(*
Nazwa:			FB_EntranceGatesFesto
Opis:			Stacja szlabanów do przesuwania formatek	
Wersja:			v1.1
Data:			2020-09-30
Autor:			DP
Urzadzenia:		do 1 szlabanu na siłowniku beckhoff i 1 szlabanu zatrzymującego na końcu
Konfiguracja:	
Info: 
*)
FUNCTION_BLOCK FB_EntranceGatesServo
VAR_INPUT
	bEnable						:BOOL;			//Zezwolenie na pracę
	bEStop						:BOOL;			//Stop Awaryjny włączony
	bRunPrepare					:BOOL;			//Rozkaz przesuwania formatek do środka 
	bRun						:BOOL;			//Rozkaz wpuszczenia dwóch formatek 
	bHoming						:BOOL;			//Zezwolenie na wykonanie bazowania i pozycjonowania podajnika
	bHeightSet					:BOOL;			//Ustaw wysokość
	bIgnoreError				:BOOL;			//Ignorowania błędów cyklu pracy
	bReset						:BOOL;			//Reset błędu, jeśli w stanie "eError"
	bBlocking					:BOOL;			//Blokowanie pierwszego szlabanu

	bOpenedGate1ActuatorSensor	:BOOL;			//Czujnik otwarcia siłownika szlabanu 1
	bOpenedGate2ActuatorSensor	:BOOL;			//Czujnik otwarcia siłownika szlabanu 2
	bClosedGate1ActuatorSensor	:BOOL;			//Czujnik zamknięcia siłownika szlabanu 1
	bClosedGate2ActuatorSensor	:BOOL;			//Czujnik zamknięcia siłownika szlabanu 2
	bMovingTwoForms				:BOOL;			//Przesuwanie o dwie formatki
	bMovingThreeForms			:BOOL;			//Przesuwanie o trzy formatki
	bManualMovement				:BOOL;			//Zezwolenie na ruchy ręcznę
	bHomingStateGate1			:BOOL;			//Stan bazowania szlabanów nr 1
	bHomingStateGate2			:BOOL;			//Stan bazowania szlabanów nr 2
	bResetState					:BOOL;			//Resetowanie stanu stacji

	//Parametry przeciągania formatek

	lrPullReadyPosition			:LREAL;			//Pozycja przeciągania przy starcie dozowania
	lrPullStopOnePhasePosition	:LREAL;			//Pozycja stopu przeciągania przy dozowaniu jednofazowym
	lrPullStopTwoPhasePosition	:LREAL;			//Pozycja stopu przeciągania przy dozowaniu dwufazowym
	lrPullVelocity				:LREAL;			//Prędkość przeciągania 
	lrPullAcceleration			:LREAL;			//Przyśpieszenie przeciągania
	lrPullDeceleration			:LREAL;			//Zwalnianie przeciągania
	
	_ALARMINFO_					:BOOL;
	iStationIndex				:UDINT;			//Numer stacji 
	sStationName				:STRING;		//Nazwa stacji

END_VAR
VAR_OUTPUT
	
	eState						:E_Station;				//Stan ogólny bloku
	eRunningState				:E_EntranceGatesState;	//Stan szlabanów
	bError						:BOOL;					//Błąd stacji	
	nErrorNr					:UDINT;					//Nr błędu podajnika platynek
	sErrorDescription			:STRING(200);			//Opis błędu
	sErrorDescription2			:STRING(200);			//Opis błędu
	sErrorStationName			:STRING;				//Nazwa stacji
	bGate1Actuator				:BOOL;					//Sterownie siłownika szlabanu 1
	bGate2Actuator				:BOOL;					//Sterownie siłownika szlabanu 2
	tCycleTime					:TIME;
	bHomingDone					:BOOL;					//Wymagane ponowne bazowanie (blad podczas bazowania lub stop awaryjny)
	bCyclePrepareDone			:BOOL;
	bCycleDone					:BOOL;
	bCycleNotDone				:BOOL;
	//WEJSCIA WYJSCIA SPRZETOWE
	nPullServoErrorNr			:UDINT;
	lrPullActualPosition		:LREAL;

END_VAR

VAR

	(**********BECKHOFF PRZECIAGANIE******************)
	mcPullMoveAbsolute			:MC_MoveAbsolute; 	// Blok nr 1 ruchu absolutnego tłoka dozownika
	mcPullManualMove			:MC_JOG;			// Blok ruchu manualnego tłokiem dozownika
	mcPullStop					:MC_Stop;			// Blok zatrzymania tłoka dozownika, jeśli to konieczne
	mcPullSoftReset				:MC_Reset;			// Blok łagodnego resetu serwa tloka dozownika
	mcPullPower					:Mc_Power;			// Blok zasilania serwa dozownika
	bPullServoPower				:BOOL; 				// Zalaczenie zasilania serwa
	// Blok resetowania twardego błędu
	fbPullHardReset				:FB_SoEReset;
	bStopped					:BOOL;
		
	// Timer blokady otwierania chwytaka
	tonOpeningGate1Blocked		:TON;
	tonOpeningGate2Blocked		:TON;
	tonClosingGate1Blocked		:TON;
	tonClosingGate2Blocked		:TON;
	tonCycleTimer				:TON;
	rtrigCycleTimerRead			:R_TRIG;	
	bLastStateGate1Actuator		:BOOL;
	bLastStateGate2Actuator		:BOOL;	
	eLastState					:E_Station;				//Stan ogólny bloku
	eLastRunningState			:E_EntranceGatesState;	//Stan podbloku
	eLastStateTemp				:E_Station;				//Stan ogólny bloku
	eLastRunningStateTemp		:E_EntranceGatesState;	//Stan podbloku

	bStateError: BOOL;
		rtPulling: R_TRIG;
	rtPreparingToReady: R_TRIG;
	rtPullingToMiddle: R_TRIG;
	tonDelayServoOn			: TON;

	bNotPreapreToReadyAfterEstop: BOOL;
	lrtest: LREAL;
	tonGate1Actuator: TON;
END_VAR

VAR_IN_OUT
	bManualGate1Actuator	:BOOL;			//Ruch ręczny siłownikiem szlabanu 1
	bManualGate2Actuator	:BOOL;			//Ruch ręczny siłownikiem szlabanu 2
	bManualPullLeft			:BOOL;			//Ruch ręczny przeciąganiem w lewo
	bManualPullRight		:BOOL;			//Ruch ręczny przeciąganiem w prawo
	PullAxisRef				:AXIS_REF;		//Struktura sterowania NC dla serwa zakręcania
END_VAR

(*Przepisywanie Homingu , rozdzielenie wyjść*)

ErrorHandling();
Control();
GatesControlBlocks();
Statistics();


(*wypracowanie sygnałów wyjściowych z bloku*)
lrPullActualPosition:=PullAxisRef.NcToPlc.ActPos;	//Pozycja 


(*Zapisywanie ostatniego stanu*)
IF eLastStateTemp<>eState THEN
	eLastState := eLastStateTemp;
END_IF
eLastStateTemp := eState;
IF eLastRunningStateTemp<>eRunningState THEN
	eLastRunningState := eLastRunningStateTemp;
END_IF
eLastRunningStateTemp := eRunningState;

(*Koniec Zapisywanie ostatniego stanu*)



IF bResetState AND NOT bBlocking THEN
	eState:=E_Station.eReady;
	eRunningState:=eLastRunningState:=E_EntranceGatesState.eReady;
	bGate1Actuator:=bHomingStateGate1;
	bGate2Actuator:=bHomingStateGate2;
END_IF

ACTION Control:

	(** TIMERY**)
	rtPulling(CLK:=eRunningState=E_EntranceGatesState.ePulling AND bOpenedGate1ActuatorSensor AND bClosedGate2ActuatorSensor, Q=>);
	rtPullingToMiddle(CLK:=eRunningState=E_EntranceGatesState.ePullingToMiddle AND bOpenedGate1ActuatorSensor AND bClosedGate2ActuatorSensor, Q=>);
	rtPreparingToReady(CLK:=eRunningState=E_EntranceGatesState.ePreparingToReady AND bClosedGate1ActuatorSensor, Q=>);
	
	tonDelayServoOn(IN:=(eState = E_Station.ePreparingToReady), PT:=T#1200MS);
	tonGate1Actuator(IN:=bGate1Actuator, PT:=T#100MS); // Opóżnienie sygnału wyjścia pierwszego szlabany, uzyte do opoznienia wylaczania drugiego
	(*****Wyłączenie enable*****)
	IF NOT bEnable THEN
		IF eState <> E_Station.eDisabled AND eState <> E_Station.ePreparingToDisable THEN
				eState 				:= E_Station.ePreparingToDisable; 
		END_IF	
	END_IF

	(*****Estop*****)
	IF NOT bEstop  THEN	
		IF eState <> E_Station.eAborted AND eState <> E_Station.eAborting AND eState <> E_Station.eDisabled THEN
				eState 				:= E_Station.eAborting; 
		END_IF
	END_IF

	
	CASE eState OF
	/////////////////////////////	
		E_Station.eDisabled: 					// Stan nieaktywnosci (Stacja wyłączona) 
		
			IF bEnable THEN
				eState 				:= E_Station.ePreparingToReady; 
			END_IF 
			
    /////////////////////////////	    
		E_Station.eAborted: 					// Stan bezpiecznego zatrzymania (po Abortingu) 

			IF bEStop THEN
				eState 				:= E_Station.ePreparingToReady;
			END_IF
			
	/////////////////////////////	
		E_Station.eAborting:                 	// Stan bezpiecznego zatrzymywania (po EStopie)

		mcPullManualMove.JogBackwards		:=	FALSE;
		mcPullManualMove.JogForward			:=	FALSE;
		mcPullMoveAbsolute.Execute 			:=	FALSE;
		
		//bPullServoPower						:=	TRUE;
		mcPullPower.Override				:=	100;		
		mcPullStop.Execute					:=	NOT bStopped;
		bNotPreapreToReadyAfterEstop		:= TRUE;
		IF (mcPullStop.Done OR mcPullStop.Error OR bStopped) THEN
			bStopped						:=	FALSE;
			bPullServoPower					:=	FALSE;
			mcPullStop.Execute				:=	FALSE;
			eLastRunningState				:=	eRunningState;
			eRunningState					:= E_EntranceGatesState.eReady;
			eState 							:=	E_Station.eAborted; 
		END_IF
			
	/////////////////////////////			
		E_Station.eError:                 	 	// Stan błędu 	
	
			mcPullMoveAbsolute.Execute 			:=	FALSE;
			mcPullStop.Execute					:= FALSE;
			IF bReset THEN
				eState 							:=	E_Station.eResetting;
			ELSE
				mcPullSoftReset	(Execute:=FALSE,Axis:=PullAxisRef);		
			END_IF
			
	/////////////////////////////
		E_Station.eResetting:					// Stan resetowania bledu (po Errorze)
			
			//Procedura obsługi resetu w zależności od błędu
			CASE nErrorNr-iStationIndex OF
		
				//Error 1 - ZACIETY SZLABAN
				1:
					bGate1Actuator								:=	FALSE;		
					nErrorNr									:=	0;
					bError										:=	FALSE;
					sErrorDescription							:=	'';		
					
				//Error 8 - SZLABANYW ZŁEJ POZYCJI			
				8: 
					bGate1Actuator								:=	FALSE;		
					bGate2Actuator								:=	TRUE;		// z 17.11.2020
				//IF tonDelayServoOn.Q THEN
					bPullServoPower								:=	TRUE;
				//END_IF
					IF bClosedGate1ActuatorSensor AND mcPullPower.Status THEN	
						mcPullMoveAbsolute.Velocity			:= lrPullVelocity;
						mcPullMoveAbsolute.Position			:= lrPullReadyPosition;
						mcPullMoveAbsolute.Acceleration		:= 15000;
						mcPullMoveAbsolute.Deceleration		:= 15000;
						mcPullMoveAbsolute.Execute			:= TRUE;
					
						//Wykonano ruch
						IF mcPullMoveAbsolute.Done THEN
							mcPullMoveAbsolute.Execute 		:=	FALSE;
							bError := FALSE;
						END_IF		
					END_IF
				//Error 9, Error 10 - BŁĄD SERWA PRZECIAGANIA
				9,10:	
					fbPullHardReset(Execute:=NOT mcPullMoveAbsolute.Execute,Axis:=PullAxisRef);
					mcPullSoftReset(Execute:=TRUE,Axis:=PullAxisRef);																		
					(*IF NOT fbPullHardReset.Busy AND NOT mcPullSoftReset.Busy AND mcPullPower.Status AND NOT PullAxisRef.Status.Error THEN
						fbPullHardReset(Execute:=FALSE,Axis:=PullAxisRef);
						mcPullSoftReset(Execute:=FALSE,Axis:=PullAxisRef);
						mcPullMoveAbsolute.Execute:=TRUE;
						mcPullMoveAbsolute.Position:=lrPullReadyPosition; 
						IF mcPullMoveAbsolute.Done=TRUE THEN
							mcPullMoveAbsolute.Execute:=FALSE;
							nErrorNr:=0;
							nPullServoErrorNr:=0;
							mcPullPower.Override:=100;
							bError := FALSE;
							sErrorDescription:='';	
						END_IF*)
					IF NOT fbPullHardReset.Busy AND NOT mcPullSoftReset.Busy (*AND NOT mcPullPower.Status*) AND NOT PullAxisRef.Status.Error  THEN
						fbPullHardReset(Execute:=FALSE,Axis:=PullAxisRef);
						mcPullSoftReset(Execute:=FALSE,Axis:=PullAxisRef);
						nPullServoErrorNr:=0;
						nErrorNr:=0;
						mcPullPower.Override:=100;
						bError := FALSE;
						sErrorDescription:='';			  	
					END_IF
					
				ELSE
					bError := FALSE;	
	
				END_CASE	
			
			IF NOT bError THEN
				nErrorNr 			:=	0;
   				sErrorDescription 	:=	'';
   				sErrorDescription2 	:=	'';	
				eState 				:=	E_Station.ePreparingToReady;
			ELSE
				eState 				:=	E_Station.eError;
			END_IF
        
	/////////////////////////////
		E_Station.eManualMovement:     			// Stan ruchów manualnych  
       
			ManualMovements();
			//Wyjście z trybu serwisowego
			IF NOT bManualMovement THEN
				
				bGate1Actuator:=bLastStateGate1Actuator;
				bGate2Actuator:=bLastStateGate2Actuator;
	
				//Ruch 
				mcPullPower.Override				:= 100;
				mcPullMoveAbsolute.Velocity			:= lrPullVelocity;
				mcPullMoveAbsolute.Position			:= lrPullReadyPosition;
				mcPullMoveAbsolute.Acceleration		:= 1000;
				mcPullMoveAbsolute.Deceleration		:= 1000;
				mcPullMoveAbsolute.Execute			:= TRUE;
			
				//Wykonano ruch
				IF mcPullMoveAbsolute.Done THEN
					mcPullMoveAbsolute.Execute 		:=	FALSE;
					eState							:=	E_Station.eReady;
					eRunningState					:=	E_EntranceGatesState.eReady;
				END_IF
				
			END_IF

	/////////////////////////////
		E_Station.eHoming:						// Stan bazowania 

			Homing();
			IF NOT bHoming AND NOT bHeightSet THEN
			   eState							:=	E_Station.ePreparingToReady;
			   mcPullManualMove.JogForward		:=	FALSE;
			   mcPullManualMove.JogBackwards	:=	FALSE;
			END_IF		
			
	/////////////////////////////
		E_Station.eHomingDone:                  // Stan wykonania bazowania 
		
			mcPullManualMove.JogForward			:=	FALSE;
			mcPullManualMove.JogBackwards		:=	FALSE;
			bHomingDone							:=	TRUE;
			IF NOT bHoming AND NOT bHeightSet THEN
			   eState:=E_Station.eReady;
			END_IF
			
	/////////////////////////////
		E_Station.ePreparingToReady:            // Stan przygotowywania do gotowosci (zawsze przed Ready)  
		
		eRunningState						:=	E_EntranceGatesState.eReady;
		IF NOT bNotPreapreToReadyAfterEstop THEN //LastRunningState przypisuje w abborting
			bGate1Actuator								:=	FALSE;		
			bGate2Actuator								:=	TRUE;		// z 17.11.2020
			IF tonDelayServoOn.Q THEN
				bPullServoPower								:=	TRUE;
			END_IF
			IF bClosedGate1ActuatorSensor AND mcPullPower.Status THEN
				IF bHomingDone THEN		
					mcPullMoveAbsolute.Velocity			:= lrPullVelocity;
					mcPullMoveAbsolute.Position			:= lrPullReadyPosition;
					mcPullMoveAbsolute.Acceleration		:= 15000;
					mcPullMoveAbsolute.Deceleration		:= 15000;
					mcPullMoveAbsolute.Execute			:= TRUE;
				
					//Wykonano ruch
					IF mcPullMoveAbsolute.Done THEN
						mcPullMoveAbsolute.Execute 		:=	FALSE;
						eRunningState					:=	E_EntranceGatesState.eReady;
						eState							:=	E_Station.eReady;	
					END_IF
								
				ELSIF NOT bHomingDone THEN
					eRunningState						:=	E_EntranceGatesState.eReady;
					eState								:=	E_Station.eReady;	
				END_IF
			END_IF
		ELSE //estop byl trakcie
			IF tonDelayServoOn.Q THEN
				bPullServoPower								:=	TRUE;
			END_IF
			IF  mcPullPower.Status THEN
				//bNotPreapreToReadyAfterEstop				:= FALSE;
				eState										:=	E_Station.eReady;	
				//eRunningState								:=	eLastRunningState; //Wpisze ostatni stan
			END_IF
		END_IF
			
	/////////////////////////////
		E_Station.ePreparingToDisable:          // Stan przygotowywania do nieaktywnosci (po wyłączeniu Enable) 
  
			bGate1Actuator							:=	FALSE;		
			bGate2Actuator							:=	FALSE;		
			bPullServoPower							:=	TRUE;
			
			IF mcPullPower.Status THEN
				mcPullPower.Override				:=	10;
				mcPullMoveAbsolute.Velocity			:=	100;
				mcPullMoveAbsolute.Execute			:=	TRUE;
				mcPullMoveAbsolute.Position			:=	lrPullReadyPosition;
				IF mcPullMoveAbsolute.Done THEN
					mcPullMoveAbsolute.Execute 		:=	FALSE;
					eState							:=	E_Station.eDisabled;
					eRunningState					:=	E_EntranceGatesState.eReady;
				END_IF	
			END_IF
			
			IF bIgnoreError THEN
				eState								:=	E_Station.eDisabled;
				eRunningState						:=	E_EntranceGatesState.eDisabled;
			END_IF
			
	/////////////////////////////
		E_Station.eReady:						// Stan gotowosci 
		
			IF (bRunPrepare OR bRun) AND NOT bCycleDone AND NOT bCycleNotDone THEN
				eState 				:= E_Station.eStarting; 
			END_IF
			IF bHoming OR bHeightSet THEN
				eState 				:= E_Station.eHoming; 
			END_IF
			IF bManualMovement THEN
				//Jeśli przejście w tryb ruchów manualnych przepisz wszystkie stany siłowników sterowanych przez moduł
				//aby zapobiec ewentualnym kolizjom po wejściu w tryb serwisowy
				bLastStateGate1Actuator		:=	bGate1Actuator;
				bLastStateGate2Actuator		:=	bGate2Actuator;
				bManualGate1Actuator		:=	bGate1Actuator;
				bManualGate2Actuator		:=	bGate2Actuator;				
				eState 						:=	E_Station.eManualMovement; 
			END_IF
			IF NOT bRun THEN
				bCycleDone 					:= FALSE;
				bCycleNotDone 				:= FALSE;	
				bCyclePrepareDone			:= FALSE;		
			END_IF
			
			bStopped						:= FALSE;
			mcPullStop.Execute				:= FALSE;
			
	/////////////////////////////
		E_Station.eStopping:					// Stan zatrzymywania 


			Running();		
			
			mcPullStop.Execute				:=	NOT bStopped;

			IF (mcPullStop.Done OR mcPullStop.CommandAborted) THEN
				 bStopped					:=	TRUE;
			END_IF
			
			IF bStopped AND NOT mcPullStop.Execute THEN
				eState 						:=	E_Station.eReady;	
			END_IF
			

	/////////////////////////////
		E_Station.eStarting:                  	// Stan uruchamiania (po Ready)
		
			eState					 := E_Station.eRunning; 
			
	/////////////////////////////
		E_Station.eRunning:               		// Stan wykonywania cyklu (po Startingu), w tym stanie osobny
 
			IF 	bNotPreapreToReadyAfterEstop THEN //Zmiana 17112020
				bNotPreapreToReadyAfterEstop := FALSE;
				eRunningState								:=	eLastRunningState; //Wpisze ostatni stan
			END_IF
		
			Running();
			IF NOT bRun AND NOT bRunPrepare THEN					(*Przerywanie cyklu*)
				eState 				 := E_Station.eStopping;	
			END_IF
			IF bCycleDone OR bCycleNotDone THEN (*Cykl zakończony*)
				//eState 				 := E_Station.eReady;//Zmiana
				eState 				 := E_Station.ePreparingToReady;
			END_IF	
			
	/////////////////////////////		
	END_CASE
END_ACTION

ACTION ErrorHandling:
//OBSŁUGA BŁĘDÓW PODAJNIKA PLATYNEK

//************LISTA BŁĘDÓW***************
bStateError:= (eState=E_Station.eError) OR (eState=E_Station.eResetting);

IF bEnable THEN

	//Error 1 - Blokada otwarcia szlabanu wejściowego nr 1
	tonOpeningGate1Blocked(IN:= bGate1Actuator AND NOT bOpenedGate1ActuatorSensor, PT:=T#2S);
	IF tonOpeningGate1Blocked.Q AND NOT bStateError THEN
		sErrorDescription:='Blokada otwarcia szlabanu wjazdowego nr 1 - sprawdź czujnik lub odblokuj mechanicznie';
		bError := TRUE;
		nErrorNr:=1;	
		nErrorNr:=nErrorNr+iStationIndex;
	END_IF
	
	//Error 2 - Blokada otwarcia szlabanu wejściowego nr 2
	tonOpeningGate2Blocked(IN:= bGate2Actuator AND NOT bOpenedGate2ActuatorSensor, PT:=T#2S);
	IF tonOpeningGate2Blocked.Q AND NOT bStateError THEN
		sErrorDescription:='Blokada otwarcia szlabanu wjazdowego nr 2 - sprawdź czujnik lub odblokuj mechanicznie';
		bError := TRUE;
		nErrorNr:=2;	
		nErrorNr:=nErrorNr+iStationIndex;
	END_IF
				
	//Error 4 - Blokada zamknięcia szlabanu wejściowego nr 1
	tonClosingGate1Blocked(IN:= NOT bGate1Actuator AND NOT bClosedGate1ActuatorSensor, PT:=T#2S);
	IF tonClosingGate1Blocked.Q AND NOT bStateError THEN
		sErrorDescription:='Blokada zamknięcia szlabanu wjazdowego nr 1 - sprawdź czujnik lub odblokuj mechanicznie';
		bError := TRUE;
		nErrorNr:=2;	
		nErrorNr:=nErrorNr+iStationIndex;
	END_IF

	//Error 5 - Blokada zamknięcia szlabanu wejściowego nr 2
	tonClosingGate2Blocked(IN:= NOT bGate2Actuator AND NOT bClosedGate2ActuatorSensor, PT:=T#2S);
	IF tonClosingGate2Blocked.Q AND NOT bStateError THEN
		sErrorDescription:='Blokada zamknięcia szlabanu wjazdowego nr 2 - sprawdź czujnik lub odblokuj mechanicznie';
		bError := TRUE;
		nErrorNr:=2;	
		nErrorNr:=nErrorNr+iStationIndex;
	END_IF	
		
(*	//Error 8 - SZLABANY W ZŁEJ POZYCJI
	IF (ABS(PullAxisRef.NcToPlc.ActPos) - lrPullReadyPosition) > 5 AND bHomingDone AND eState = E_Station.eReady AND NOT bResetState AND NOT bStateError THEN
		bError := TRUE;
		nErrorNr:=8;
		nErrorNr:=nErrorNr+iStationIndex;
		nPullServoErrorNr:=PullAxisRef.Status.ErrorID;
		sErrorDescription:='Szlabany w złej pozycji, zresetuj';
		sErrorDescription2:=INT_TO_STRING(LREAL_TO_INT(PullAxisRef.NcToPlc.ActPos));
	END_IF;	*)
	
	//Error 9 - BŁĄD SERWA PODNOSZENIA ZAKRĘCARKI
	IF (PullAxisRef.Status.Error OR mcPullPower.Error) AND NOT bStateError THEN
		bError := TRUE;
		nErrorNr:=9;
		nErrorNr:=nErrorNr+iStationIndex;
		nPullServoErrorNr:=PullAxisRef.Status.ErrorID;
		sErrorDescription:='Błąd napędu przeciągania Błąd NC:';
		sErrorDescription2:=F_AxErrMsg(nPullServoErrorNr);
	END_IF;	
	
	//Error 10 - BŁĄD INNY SERWA PODNOSZENIA ZAKRĘCARKI
	IF  mcPullMoveAbsolute.Error AND NOT bStateError THEN
		bError := TRUE;
		nErrorNr:=10;
		nErrorNr:=nErrorNr+iStationIndex;
		nPullServoErrorNr:=mcPullMoveAbsolute.ErrorID;
		sErrorDescription:='Błąd napędu przeciągania Błąd NC:';
		sErrorDescription2:=F_AxErrMsg(nPullServoErrorNr);
	END_IF;
	
	
	
ELSE
	bError := FALSE;
END_IF
	
//*******KONIEC LISTA BŁĘDÓW***************	

	

//******************PRZEJŚCIE DO eERROR*****************************

IF bError AND NOT bStateError THEN
	IF eLastState = eRunning THEN
		bCycleNotDone := TRUE;
	END_IF
	eState := E_Station.eError;
END_IF

//****************WYŚWIETLANIE STATUSU BLEDU***********************


(*Wyświetlanie błedu na wyjściu*)
bError;

(*Przepisywanie nazwy stacji*)
sErrorStationName:=sStationName;
END_ACTION

ACTION GatesControlBlocks:
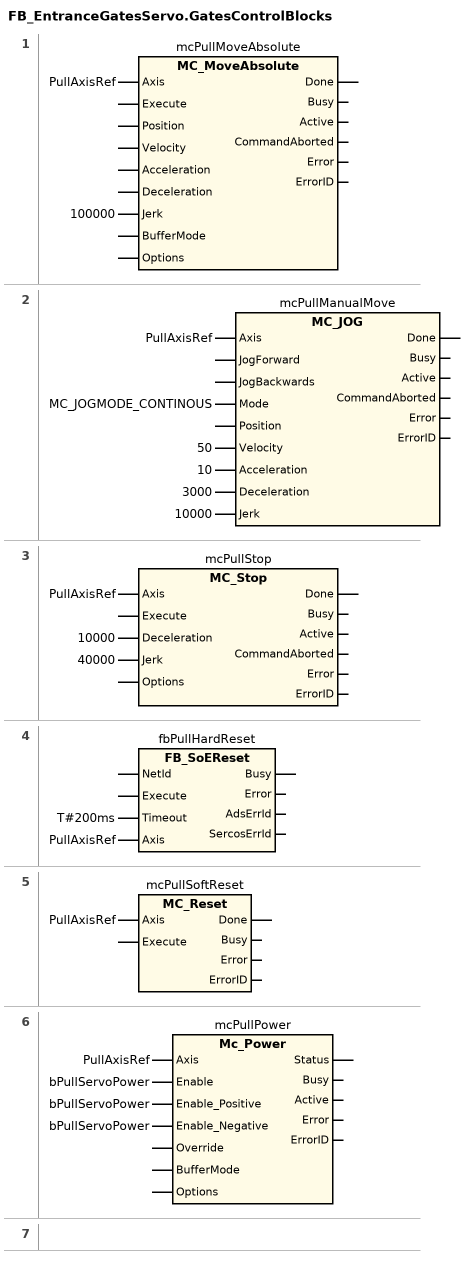
// NETWORK 1
mcPullMoveAbsolute(Axis := PullAxisRef, Jerk := 100000); // MC_MoveAbsolute

// NETWORK 2
mcPullManualMove(
    Axis := PullAxisRef,
    Mode := MC_JOGMODE_CONTINOUS,
    Velocity := 50,
    Acceleration := 10,
    Deceleration := 3000,
    Jerk := 10000); // MC_JOG

// NETWORK 3
mcPullStop(Axis := PullAxisRef, Deceleration := 10000, Jerk := 40000); // MC_Stop

// NETWORK 4
fbPullHardReset(Timeout := T#200ms, Axis := PullAxisRef); // FB_SoEReset

// NETWORK 5
mcPullSoftReset(Axis := PullAxisRef); // MC_Reset

// NETWORK 6
mcPullPower(
    Axis := PullAxisRef,
    Enable := bPullServoPower,
    Enable_Positive := bPullServoPower,
    Enable_Negative := bPullServoPower); // Mc_Power

// NETWORK 7
END_ACTION

ACTION Homing:
//Ustawienia początkowe
bGate1Actuator						:=	FALSE;
bGate2Actuator						:=	TRUE;

//Włączanie zasilania
mcPullPower.Override				:=	100;
mcPullManualMove.JogBackwards		:=	FALSE;
mcPullManualMove.JogForward			:=	FALSE;
bPullServoPower						:=	TRUE;

//Serwo włączone
IF mcPullPower.Status THEN
	
	//Ruch 
	mcPullMoveAbsolute.Velocity			:= lrPullVelocity;
	mcPullMoveAbsolute.Position			:= lrPullReadyPosition;
	mcPullMoveAbsolute.Acceleration		:= 1000;
	mcPullMoveAbsolute.Deceleration		:= 1000;
	mcPullMoveAbsolute.Execute			:= TRUE;

	//Wykonano ruch
	IF mcPullMoveAbsolute.Done THEN
		mcPullMoveAbsolute.Execute 		:=	FALSE;
		eState							:=	E_Station.eHomingDone;
	END_IF
END_IF
END_ACTION

ACTION ManualMovements:

//W trybie ruchów manualnych wykonuj ruchy za pomocą rozkazów manualnych
IF NOT bRun AND NOT bRunPrepare THEN
	bGate1Actuator					:=	bManualGate1Actuator;
	bGate2Actuator					:=	bManualGate2Actuator;	
	mcPullPower.Override			:=	100;
	mcPullManualMove.JogForward		:=	bManualPullRight;
	mcPullManualMove.JogBackwards	:=	bManualPullLeft;
ELSE	
	;
END_IF


IF bHoming OR bHeightSet THEN
	eState:=E_Station.eHoming;
END_IF
	

Running();


IF NOT bRun AND NOT bRunPrepare THEN
	bCycleDone 					:= FALSE;
	bCycleNotDone 				:= FALSE;			
	bCyclePrepareDone			:= FALSE;
END_IF
END_ACTION

ACTION Running:


CASE eRunningState OF
	
	//NIEGOTOWY
	E_EntranceGatesState.eDisabled:
			eRunningState:=E_EntranceGatesState.eReady;
		
	//ZGRZEWANIE GOTOWY DO PRACY
	E_EntranceGatesState.eReady:
		
		//Jeśli komenda podania platynki przejdź do stanu zasysania platynki
		IF NOT bCycleDone AND NOT bCycleNotDone THEN
			IF bBlocking THEN
				eRunningState := E_EntranceGatesState.eBlocking;	
			ELSIF bRun THEN
				eRunningState:=E_EntranceGatesState.ePulling;
			ELSIF bRunPrepare THEN
				eRunningState:=E_EntranceGatesState.ePullingToMiddle;				
			END_IF
		END_IF

	//Przesuwanie do środka (przyśpieszenie cyklu*)
	E_EntranceGatesState.ePullingToMiddle:
		
		bGate1Actuator:=TRUE;
		IF tonGate1Actuator.Q THEN //LU205
			bGate2Actuator:=FALSE;
		END_IF
		IF bOpenedGate1ActuatorSensor AND bClosedGate2ActuatorSensor THEN
			mcPullMoveAbsolute.Velocity			:=	lrPullVelocity;
			mcPullMoveAbsolute.Position			:=	lrPullStopOnePhasePosition/3;	
			mcPullMoveAbsolute.Acceleration		:=	lrPullAcceleration;
			mcPullMoveAbsolute.Deceleration		:=	lrPullDeceleration;
			IF rtPullingToMiddle.Q THEN
				mcPullMoveAbsolute.Execute		:=	TRUE;
			END_IF
			//Wykonano ruch
			IF mcPullMoveAbsolute.Done AND (lrPullActualPosition>mcPullMoveAbsolute.Position-6 AND lrPullActualPosition<mcPullMoveAbsolute.Position+6) THEN
				mcPullMoveAbsolute.Execute		:=	FALSE;
				eRunningState					:=	E_EntranceGatesState.ePullingToMiddleDone;			
			END_IF
		END_IF		

	//Koniec przesuwanie do środka (przyśpieszenie cyklu*)
	E_EntranceGatesState.ePullingToMiddleDone:	
		bCyclePrepareDone						:=	TRUE;
		IF bRun THEN
			eRunningState						:=	E_EntranceGatesState.ePulling; 
		END_IF
		
	//Rozpoczynanie przeciąganai
	E_EntranceGatesState.ePulling:
		
		bGate1Actuator:=TRUE;
		IF tonGate1Actuator.Q THEN //LU205
			bGate2Actuator:=FALSE;
		END_IF
		IF bOpenedGate1ActuatorSensor AND bClosedGate2ActuatorSensor THEN
		//Wpisanie przyśpieszeń przeciągania
			mcPullMoveAbsolute.Velocity			:=	lrPullVelocity;
			IF bMovingTwoForms AND bMovingThreeForms THEN 	(*przesuwanie do pozycji końcowej, trzy formatki*)
				mcPullMoveAbsolute.Position		:=	lrPullStopOnePhasePosition;
			ELSIF bMovingTwoForms THEN						(*przesuwanie do pozycji prawie końcowej, dwie formatki*)
				mcPullMoveAbsolute.Position		:=	(((lrPullStopOnePhasePosition-lrPullReadyPosition)*2/3)+lrPullReadyPosition);
			ELSE
				mcPullMoveAbsolute.Position		:=	lrPullStopTwoPhasePosition;
			END_IF	
			mcPullMoveAbsolute.Acceleration		:=	lrPullAcceleration;
			mcPullMoveAbsolute.Deceleration		:=	lrPullDeceleration;
			IF rtPulling.Q THEN
				mcPullMoveAbsolute.Execute		:=	TRUE;
			END_IF

			//Zamykanie szlabanu troche wcześniej
			IF  mcPullMoveAbsolute.Position - lrPullActualPosition < 100 THEN
				bGate2Actuator	:=	TRUE;
			END_IF
			
			//Wykonano ruch			
			IF mcPullMoveAbsolute.Done  AND lrPullActualPosition>mcPullMoveAbsolute.Position-3 AND lrPullActualPosition<mcPullMoveAbsolute.Position+3 THEN
				mcPullMoveAbsolute.Execute		:=	FALSE;
				eRunningState					:=	E_EntranceGatesState.ePullingDone;			
			END_IF
		END_IF
		
	//Koniec przeciągania
	E_EntranceGatesState.ePullingDone:
			bGate1Actuator	:=	FALSE;
			bGate2Actuator	:=	TRUE;
			IF bClosedGate1ActuatorSensor THEN
				bCycleDone		:=	TRUE;
				eRunningState:=E_EntranceGatesState.eReady; 
			END_IF

	//Blokowanie
	E_EntranceGatesState.eBlocking:
		bGate1Actuator:=FALSE;
		bGate2Actuator:=TRUE;
		IF (NOT bBlocking) OR (NOT bEnable) THEN 
			eRunningState:=E_EntranceGatesState.eReady;
		END_IF
		
END_CASE
END_ACTION

ACTION Statistics:



rtrigCycleTimerRead(CLK:=eRunningState=E_EntranceGatesState.eReady);
IF rtrigCycleTimerRead.Q THEN
	tCycleTime:=tonCycleTimer.ET;
END_IF
tonCycleTimer(IN:=eRunningState>E_EntranceGatesState.eReady,PT:=T#1D);
END_ACTION

END_FUNCTION_BLOCK

(* stored: Version 1.1.0.1, ProductVersion 3.1.4026.13, FileIdentifier ca9160cc29483d8e053615e014315919c6afe09b, FileSignature 25ea37506f2cd35d89080a3221106e9b58b4cd28ac8e41dd3bfe31819c84fc4835c4c917f95bb1e7dfab556e839eeb1fdda5594818283215559957610ada4c129db27689f54c9771cafb1a1440c170f8dea240f02a4125de1a3aada6e3039d3c9cf6b9f413c1a6994d84fedca6a17edb7668fe7832647d2779973957e8ee82b784e2fb5744907e74a69dd241d0e74955935fb51487896f6823d15ddb80fc3ecf64d894758565535977b5722dbea1a94378471390048c7148ea3ada65400168f3f5b1e6c35b5cd04b1428edf80d3553daf01b1523f83c4ca0919fd4e289eb0e870f8afd1bbeaf0f4869767e208d3e684eba9d048bc29e33ebbcfb75e3c509fffe
   POU FB_EntranceGatesServo: Id {bbda39e3-4c1e-45a2-b62d-875cf3179e4e}, SpecialFunc None
   Action Control: Id {a9cc0879-069f-4b25-b0e1-f8e0188450db}
   Action ErrorHandling: Id {7f91051d-649d-4178-9e0b-25156a3ae81e}
   Action GatesControlBlocks: Id {a899135a-62f0-4b6e-94cb-d740e3a255ef}
   Action Homing: Id {3b46685b-cfc9-4711-84e1-92ad55d6470e}
   Action ManualMovements: Id {b6312e4c-4f5d-4815-9390-5f750d7253ee}
   Action Running: Id {32557882-ee8e-4409-bc77-9b073f2a5f8d}
   Action Statistics: Id {74c13e8b-919f-40dd-ad8d-b3614f1e729c} *)
